Staubli VAL3: getNextID.pgx

public program getNextID(num& x_nNextID[])
begin
  // This program checks if there is an object in the queue
  //
  // Output Param
  //  x_nNextID : value of the next object ID in the queue
  //        <0 --> No object available
  //
  //
  //----------------------------------------------------------------
  //
  setMutex(bLockQueueAcces)
  //
  if (nQueueID[nIdxPull]>=0)
    x_nNextID=nQueueID[nIdxPull]
    // mark the object as "in use"
    if (round(nNumbOfUser[nIdxPull])==0)
      call setObjectInUse(nIdxPull)
    endIf
  else
    x_nNextID=-1
  endIf
  //
  bLockQueueAcces=false
end
